// Block: PPrgArchive2

DATA_BLOCK PPrgArchive2
VERSION : 0.1
   NON_RETAIN
   VAR
      PRG : Array[101..200] of PPrg_Data;
   END_VAR

BEGIN
   // No initialization required
END_DATA_BLOCK
